// TIA Portal project "Analog Input" (V17)

(* hardware
DEVICE "S7-1200 station_1"  S7-1200 Station
   slot 0: "Rack_0"  S7-1200 Rack  Rack  V1.0
   slot 1: "Analog Input 0-10VDC/4-12mA"  CPU 1214C DC/DC/DC  6ES7 214-1AG40-0XB0  V4.5
*)

// ===== PLC "Analog Input 0-10VDC/4-12mA"  CPU 1214C DC/DC/DC =====

VAR_GLOBAL   // PLC tag table "Default tag table"
   "Blue_Light" AT %Q0.0 : Bool;
   "Stop button (NC)" AT %I0.0 : Bool;
   "Red_Light" AT %Q0.4 : Bool;
   "Yellow_Light" AT %Q0.5 : Bool;
   "Green_Light" AT %Q0.6 : Bool;
   "White_Light" AT %Q0.7 : Bool;
   "AlwaysTRUE" AT %M1.2 : Bool;
   "AlwaysFALSE" AT %M1.3 : Bool;
   "Clock_Byte" AT %MB0 : Byte;
   "Clock_10Hz" AT %M0.0 : Bool;
   "Clock_5Hz" AT %M0.1 : Bool;
   "Clock_2.5Hz" AT %M0.2 : Bool;
   "Clock_2Hz" AT %M0.3 : Bool;
   "Clock_1.25Hz" AT %M0.4 : Bool;
   "Clock_1Hz" AT %M0.5 : Bool;
   "Clock_0.625Hz" AT %M0.6 : Bool;
   "Clock_0.5Hz" AT %M0.7 : Bool;
   "SR01" AT %M2.0 : Bool;
   "Reset_up" AT %M2.1 : Bool;
   "System_Byte" AT %MB1 : Byte;
   "Start Button" AT %I0.1 : Bool;
   "Buzzer" AT %Q1.1 : Bool;
   "Analog_In_Ch0" AT %IW64 : Word;
   "Running" AT %M3.2 : Bool;
   "Start_done" AT %M3.1 : Bool;
   "Starting" AT %M3.0 : Bool;
   "Run_Mode" AT %MB2 : Byte;
END_VAR

DATA_BLOCK "Norm_Scale_DB"   // DB1
{ S7_Optimized_Access := 'TRUE' }
VERSION : 0.1
// stored: InstanceOfName Norm_Scale
"Norm_Scale"
BEGIN
END_DATA_BLOCK

DATA_BLOCK "Main_DB"   // DB2
{ S7_Optimized_Access := 'TRUE' }
VERSION : 0.1
   VAR
      Q25 : Bool;
      Q50 : Bool;
      Q75 : Bool;
      Q100 : Bool;
      AI_Buffer : Word;
   END_VAR
BEGIN
END_DATA_BLOCK

FUNCTION_BLOCK "Norm_Scale"   // FB1, LAD
{ S7_Optimized_Access := 'TRUE' }
VERSION : 0.1
   VAR_INPUT
      AI0 : Int;
      min_normx : Int;
      min_scalex : Int;
      max_normx : Int;
      max_scalex : Int;
   END_VAR
   VAR_OUTPUT
      AIQ : Real;
   END_VAR
   VAR_TEMP
      norm_scale : Real;
   END_VAR
BEGIN

REGION Network 1
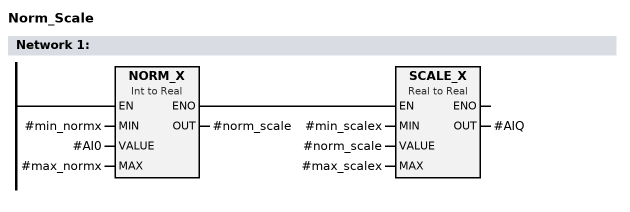
   RUNG wire#powerrail
      { S7_Templates := "[SrcType := Int, DestType := Real]" } Normalize(min := #min_normx, value := #AI0, max := #max_normx, out => #norm_scale)
      { S7_Templates := "[SrcType := Real, DestType := Real]" } Scale(min := #min_scalex, value := #norm_scale, max := #max_scalex, out => #AIQ)
   END_RUNG
   // the same network as SCL:
   #norm_scale := NORM_X(MIN := #min_normx, VALUE := #AI0, MAX := #max_normx);
   #AIQ := SCALE_X(MIN := #min_scalex, VALUE := #norm_scale, MAX := #max_scalex);
END_REGION
END_FUNCTION_BLOCK

ORGANIZATION_BLOCK "Main"   // OB1, LAD, ProgramCycle
TITLE = "Main Program Sweep (Cycle)"
{ S7_Optimized_Access := 'TRUE' }
VERSION : 0.1
// Author: Andi Sama
// Organization: Sinergi Wahana Gemilang
// Date (created): Jan 6, 2023
// Date (last modified): Jan 16, 2023
// 
// Purpose: Understanding 0-10VDC/4-20mA Analog Signal
// - Real PLC: Siemens PLC 1200 DC/DC/DC
// 
// Special note:
// As the Siemens S7-1200 PLC only support 0-10V voltage signaling for its analog input, a 500 Ohm resistor with very low tolerance (e.g. 0.1%) needs to be installed in paralel to analog input in order to receive 4-20mA. Otherwise the default is to receive only 0-10V.
// See details in: https://support.industry.siemens.com/cs/ww/en/view/67396370.
// 
// Start - Blue light ON
// 
// One of the following:
// 
// 1. Voltage
// Analog Input 0-2.5VDC Red light ON
// Analog Input 2.5-5VDC -  Yellow light ON
// Analog Input 5-7.5VDC -  Green light ON
// Analog Input 75-10VDC -  White light ON
// 
// 2. Current
// Analog Input 0-25mA -  Red light ON
// Analog Input 25-50mA -  Yellow light ON
// Analog Input 50-75mA -  Green light ON
// Analog Input 75-100mA -  White light ON
   VAR_INPUT
      Initial_Call : Bool;   // Initial call of this OB
      Remanence : Bool;   // =True, if remanent data are available
   END_VAR
   VAR_TEMP
      Ch0AQ1 : Bool;
      Ch0AQ0 : Bool;
      Ch0AI0 : Bool;
      Ch0_Normalized_Scaled : Real;
      Start : Bool;
      Start_done : Bool;
      PLC_Initialized : Bool;
   END_VAR
   VAR CONSTANT
      AI_Lowest : Real := 4.0;
      AI_Low : Real := 8.0;
      AI_Mid : Real := 12.0;
      AI_High : Real := 16.0;
      AI_Highest : Real := 20.0;
      PLC_ADC_Max : Int := 27648;
   END_VAR
   VAR_TEMP   // added for the SCL form of the ladder/FBD networks
      _w1 : Bool;
   END_VAR
BEGIN

REGION Network 1: Preparation
   // Real PLC
   // - Directly gets analog input (0-10VDC or 4-20mA) from PLC Analog Input (CH00)
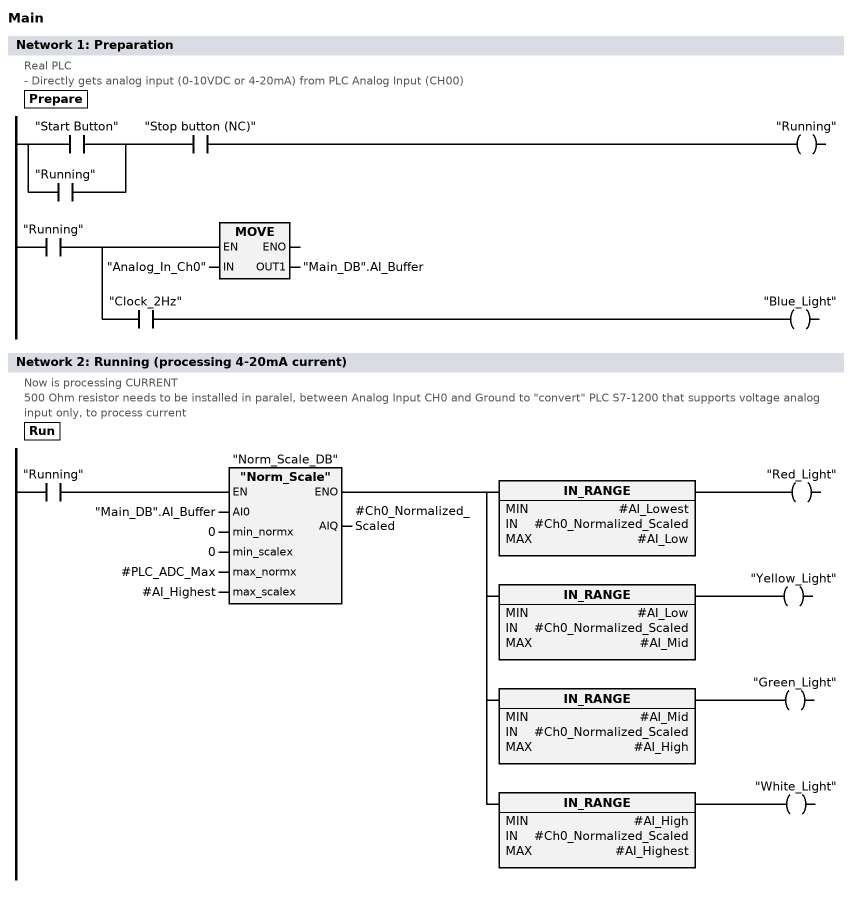
   Label( Prepare )
   RUNG wire#powerrail
      Contact( "Start Button" )
      wire#w1
      Contact( "Stop button (NC)" )
      Coil( "Running" )
   END_RUNG
   RUNG wire#powerrail
      Contact( "Running" )
   END_RUNG wire#w1
   RUNG wire#powerrail
      Contact( "Running" )
      wire#w2
      Move(in := "Analog_In_Ch0", out1 => "Main_DB".AI_Buffer)
   END_RUNG
   RUNG wire#w2
      Contact( "Clock_2Hz" )
      Coil( "Blue_Light" )
   END_RUNG
   // the same network as SCL:
   Prepare:
   "Running" := ("Start Button" OR "Running") AND "Stop button (NC)";
   IF "Running" THEN "Main_DB".AI_Buffer := "Analog_In_Ch0"; END_IF;
   "Blue_Light" := "Running" AND "Clock_2Hz";
END_REGION

REGION Network 2: Running (processing 4-20mA current)
   // Now is processing CURRENT
   // 500 Ohm resistor needs to be installed in paralel, between Analog Input CH0 and Ground to "convert" PLC S7-1200 that supports voltage analog input only, to process current
   Label( Run )
   RUNG wire#powerrail
      Contact( "Running" )
      "Norm_Scale_DB"(AI0 := "Main_DB".AI_Buffer, min_normx := 0, min_scalex := 0, max_normx := #PLC_ADC_Max, max_scalex := #AI_Highest, AIQ => #Ch0_Normalized_Scaled)
      wire#w1
      { S7_Templates := "SrcType := Real" } InRange(min := #AI_Lowest, in := #Ch0_Normalized_Scaled, max := #AI_Low)
      Coil( "Red_Light" )
   END_RUNG
   RUNG wire#w1
      { S7_Templates := "SrcType := Real" } InRange(min := #AI_Low, in := #Ch0_Normalized_Scaled, max := #AI_Mid)
      Coil( "Yellow_Light" )
   END_RUNG
   RUNG wire#w1
      { S7_Templates := "SrcType := Real" } InRange(min := #AI_Mid, in := #Ch0_Normalized_Scaled, max := #AI_High)
      Coil( "Green_Light" )
   END_RUNG
   RUNG wire#w1
      { S7_Templates := "SrcType := Real" } InRange(min := #AI_High, in := #Ch0_Normalized_Scaled, max := #AI_Highest)
      Coil( "White_Light" )
   END_RUNG
   // the same network as SCL:
   Run:
   "Norm_Scale_DB"(EN := "Running",   // "Norm_Scale"
                   AI0 := "Main_DB".AI_Buffer,
                   min_normx := 0,
                   min_scalex := 0,
                   max_normx := #PLC_ADC_Max,
                   max_scalex := #AI_Highest,
                   AIQ => #Ch0_Normalized_Scaled,
                   ENO => #_w1);
   "Red_Light" := #_w1 AND (#AI_Lowest <= #Ch0_Normalized_Scaled) AND (#Ch0_Normalized_Scaled <= #AI_Low);
   "Yellow_Light" := #_w1 AND (#AI_Low <= #Ch0_Normalized_Scaled) AND (#Ch0_Normalized_Scaled <= #AI_Mid);
   "Green_Light" := #_w1 AND (#AI_Mid <= #Ch0_Normalized_Scaled) AND (#Ch0_Normalized_Scaled <= #AI_High);
   "White_Light" := #_w1 AND (#AI_High <= #Ch0_Normalized_Scaled) AND (#Ch0_Normalized_Scaled <= #AI_Highest);
END_REGION
END_ORGANIZATION_BLOCK

ORGANIZATION_BLOCK "Initialization"   // OB100, LAD, Startup
TITLE = "Complete Restart"
{ S7_Optimized_Access := 'TRUE' }
VERSION : 0.1
   VAR_INPUT
      LostRetentive : Bool;   // True if retentive data are lost
      LostRTC : Bool;   // True if date and time are lost
   END_VAR
BEGIN

REGION Network 1: Start
   // Select one of Run Modes:
   // 1: Real PLC 
   // 2: PLC Simulator
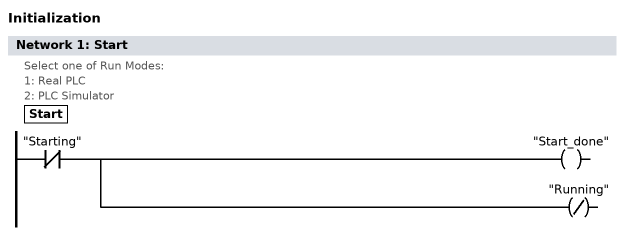
   Label( Start )
   RUNG wire#powerrail
      I_Contact( "Starting" )
      wire#w1
      Coil( "Start_done" )
   END_RUNG
   RUNG wire#w1
      I_Coil( "Running" )
   END_RUNG
   // the same network as SCL:
   Start:
   "Start_done" := NOT "Starting";
   "Running" := NOT (NOT "Starting");
END_REGION
END_ORGANIZATION_BLOCK